(* CODESYS project CtaVisUser_1.0.0.0.library
   DocFormat: reStructuredText
   DefaultNamespace: CtaVisUser
   Version: 1.0.0.0
   Placeholder: CtaVisUser
   Company: CTA
   Description: Visu User Library der CTA
   CompiledLibraryCompatibilityVersion: CODESYS V3.5 SP16 Patch 3
   LanguageModelAttribute: qualified-access-only
   Title: CtaVisUser
   Author: SIS

Project tree, tasks and I/O mapping:
  libraries: CmpBitmapPool, 3.5.17.0 (System); Visu Utils, 4.5.0.0 (System); Standard, 3.5.18.0 (System); VisuElemBase, * (System); VisuUserMgmt, * (System); VisuDialogs, * (System); VisuSymbols, 4.5.0.0 (System); CtaVisSymbols, 1.0.0.0 (CTA)
  40 Visualizations/
    visualisation VIS_USER
    visualisation DIA_USER_MANAGEMENT
  30 Program Organization Units/
  00000000-0000-0000-0000-000000000000|D:\CoDeSys\LibrariesV3\trunk\Intern\CAA\CAA Template\3.4.0.0 draft\Placeholder.xml
  00000000-0000-0000-0000-000000000000|D:\CoDeSys\LibrariesV3\trunk\Intern\CAA\CAA Template\3.2.0.3 draft\Prefix.pdf
  00000000-0000-0000-0000-000000000000|D:\CoDeSys\LibrariesV3\trunk\Intern\CAA\CAA Template\3.5.2.0 draft\Placeholder.xml
  20 Structs/
  50 Images/
  10 Documenation/
    global variables VersionHistory
    global variables readMe
  21 Interface/
  11 Library Parameter/
  12 Konstanten/
  60 Textlisten/
  13 Globale Variablen/
  5ce3da45-db07-42e7-a21c-a00fff4ed8f6|Icons\alert.svg
  5ce3da45-db07-42e7-a21c-a00fff4ed8f6|Icons\arrow-down.svg
  5ce3da45-db07-42e7-a21c-a00fff4ed8f6|Icons\arrow-down_square.svg
  5ce3da45-db07-42e7-a21c-a00fff4ed8f6|Icons\arrow-left_solo_black.svg
  5ce3da45-db07-42e7-a21c-a00fff4ed8f6|Icons\arrow-right_solo_black.svg
  5ce3da45-db07-42e7-a21c-a00fff4ed8f6|Icons\arrow-up.svg
  5ce3da45-db07-42e7-a21c-a00fff4ed8f6|Icons\calendar-range.svg
  5ce3da45-db07-42e7-a21c-a00fff4ed8f6|Icons\check.svg
  5ce3da45-db07-42e7-a21c-a00fff4ed8f6|Icons\clock-outline.svg
  5ce3da45-db07-42e7-a21c-a00fff4ed8f6|Icons\close_solo_black.svg
  5ce3da45-db07-42e7-a21c-a00fff4ed8f6|Icons\CtaInfo.svg
  5ce3da45-db07-42e7-a21c-a00fff4ed8f6|Icons\database_black.svg
  5ce3da45-db07-42e7-a21c-a00fff4ed8f6|Icons\delete_solo_black.svg
  5ce3da45-db07-42e7-a21c-a00fff4ed8f6|Icons\engine.svg
  5ce3da45-db07-42e7-a21c-a00fff4ed8f6|Icons\front_hand_Black.svg
  5ce3da45-db07-42e7-a21c-a00fff4ed8f6|Icons\front_hand_Yellow_Off.svg
  5ce3da45-db07-42e7-a21c-a00fff4ed8f6|Icons\gear.svg
  5ce3da45-db07-42e7-a21c-a00fff4ed8f6|Icons\home.svg
  5ce3da45-db07-42e7-a21c-a00fff4ed8f6|Icons\information-variant.svg
  5ce3da45-db07-42e7-a21c-a00fff4ed8f6|Icons\lightning-bolt-circle.svg
  5ce3da45-db07-42e7-a21c-a00fff4ed8f6|Icons\message.svg
  5ce3da45-db07-42e7-a21c-a00fff4ed8f6|Icons\message-alert-variant.svg
  5ce3da45-db07-42e7-a21c-a00fff4ed8f6|Icons\minus_solo_black.svg
  5ce3da45-db07-42e7-a21c-a00fff4ed8f6|Icons\plus_solo_black.svg
  5ce3da45-db07-42e7-a21c-a00fff4ed8f6|Icons\power_solo_black.svg
  5ce3da45-db07-42e7-a21c-a00fff4ed8f6|Icons\refresh_solo_black.svg
  5ce3da45-db07-42e7-a21c-a00fff4ed8f6|Icons\SearchFilter.svg
  5ce3da45-db07-42e7-a21c-a00fff4ed8f6|Icons\signal-celular-alt.svg
  5ce3da45-db07-42e7-a21c-a00fff4ed8f6|Icons\toggle-switch.svg
  5ce3da45-db07-42e7-a21c-a00fff4ed8f6|Icons\Modbus_Organization_Logo.svg
  5ce3da45-db07-42e7-a21c-a00fff4ed8f6|Icons\CheckboxUnchecked_withe.svg
  5ce3da45-db07-42e7-a21c-a00fff4ed8f6|Icons\lock_open_black.svg
  5ce3da45-db07-42e7-a21c-a00fff4ed8f6|Icons\check_green.svg
  5ce3da45-db07-42e7-a21c-a00fff4ed8f6|Icons\filter_black.svg
  5ce3da45-db07-42e7-a21c-a00fff4ed8f6|Icons\CtaLogo.png
  5ce3da45-db07-42e7-a21c-a00fff4ed8f6|Icons\Grafana_Logo.svg
  5ce3da45-db07-42e7-a21c-a00fff4ed8f6|Icons\hourglass_top.svg
  text list GlobalTextList
*)

// 10 Documenation/VersionHistory
(* 

.. image:: ../../Images/CTA_Logo.jpg
   :align: right
   :width: 15% 

**Vorlage**   


============ =========== =========== ============================================
**Date**     **Version** **Author**  **Change**
------------ ----------- ----------- --------------------------------------------
04.03.2021   0.0.0.0     SIS         Vorlage erstellt

============ =========== =========== ============================================


*)
VAR_GLOBAL
    stInfo : STRING:= '0.0.0.0, Vorlage, CTA';
END_VAR

// 10 Documenation/readMe
(*

**ReadMe**
 
|	**Empfehlung**
|
|	Dokumentrieren Sie die Library für eine nachhaltige Entwicklung
|     
| *Beispiel*
| 
| Dies ist die Vorlage Library der CTA. Erstellen Sie ihre Library anhand dieser Vorlage.
*)

VAR_GLOBAL
    xReadMeDone              :   BOOL;
END_VAR

// 40 Visualizations/VIS_USER
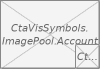
VISUALIZATION VIS_USER  // 100x69
    Image (0,0 100x69), image: CtaVisSymbols.ImagePool.Account
        OnMouseClick:  Dialog=DIA_USER_MANAGEMENT, OpenModal=True, OpenCentered=True
    Image (75,44 25x25), image: CtaVisSymbols.ImagePool.check_green
        OnMouseClick:  Dialog=DIA_USER_MANAGEMENT, OpenModal=True, OpenCentered=True
END_VISUALIZATION

// 40 Visualizations/DIA_USER_MANAGEMENT
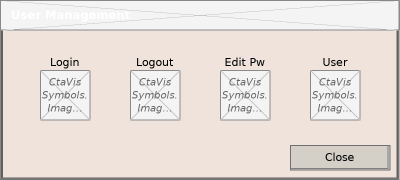
VISUALIZATION DIA_USER_MANAGEMENT  // 400x180
    Rectangle (0,0 399x180)
    Image (40,70 50x50), image: CtaVisSymbols.ImagePool.lock_open_black
        OnMouseClick:  Type=Login
    Image (130,70 50x50), image: CtaVisSymbols.ImagePool.lock_closed_black
        OnMouseClick:  Type=Logout
    Image (310,70 50x50), image: CtaVisSymbols.ImagePool.Settings+
        OnMouseClick:  Type=OpenUserConfiguration
    Image (220,70 50x50), image: CtaVisSymbols.ImagePool.Edit_Stift
        OnMouseClick:  Type=ChangeUserPassword
    Label (40,55 50x15), "Login"
    Label (130,55 50x15), "Logout"
    Label (220,55 50x15), "Edit Pw"
    Label (310,55 50x15), "User"
    Image (0,0 400x30), "User Management", image: VisuDialogs.ImagePoolDialogs.Title
    Button (290,145 100x25), "Close"
        OnMouseClick:  Dialog=Current Dialog, Result=OK, NumpadKeypadSet=True
END_VISUALIZATION
